{attribute 'qualified_only'}
VAR_GLOBAL
	gSimulation : BOOL;
	gDeklCount : INT;
	gFBInitCount : UDINT;
	gInstanceIDCount : UDINT;
END_VAR

(* stored: Version 1.1.0.1, ProductVersion 3.1.4020.12
   GVL GVL: Id {4766361d-2c6f-42f1-a9cf-270d901037db} *)
